FUNCTION_BLOCK TmsEmbarkStation EXTENDS Process IMPLEMENTS ITF_SwitchStation
VAR_INPUT
	StateMachine : IPmlStateMachine;
	TmsSwitch : ITF_TmsSwitch;
END_VAR
VAR_OUTPUT
END_VAR
VAR
	DepartMover : ITmsMover;
	_stationPosition : INT := 1; //1 is low, 2 is high
	State :(
		Init,                                               
		Ready,                                 
        Waiting,
		Processing,
		Register,
		Boarding,
		BoardingComplete,
		Moving); 
	_switchPosition: MC_LREAL;
	demandPosition : SwitchState;
END_VAR

CASE State OF
	Init:
		_Operating := _Clear := _Complete := _Ready := _HasMover := FALSE;
		_Positions[1] := _Positions[2] := _Positions[3] := _Positions[4] := 0;
		NumberOfPositions := 0;
		AssignedPositions := 1;
		StationMovers := 0;
		State := Ready;
	
	Ready:	
		IF StateMachine.GetCurrentState() = E_PMLState.ePMLState_Clearing THEN
			_Operating := _Complete := _HasMover := FALSE;
			_Clear := _Ready := TRUE;
			StationMovers := 0;
			State := Waiting;
		END_IF
	
	Waiting:
		IF _HasMover THEN
			State := Processing;
			_Operating := TRUE;
			_Clear := FALSE;
			_Ready := FALSE;
			_Complete := FALSE;
		END_IF
		
	Processing:
		IF _stationPosition = 1 THEN
			IF TmsSwitch.Switch = SwitchState.Down THEN
				IF DepartMover.ActiveTrack = 16#01010790 THEN
					State := Register;
				ELSE
					DepartMover.ActivateTrack(16#01010790);
					State := Register;
				END_IF
				demandPosition := SwitchState.Middle;
			ELSIF TmsSwitch.Switch = SwitchState.Middle THEN
				IF DepartMover.ActiveTrack = 16#010100E0 THEN
					State := Register;
				ELSE
					DepartMover.ActivateTrack(16#010100E0);
					State := Register;
				END_IF
				demandPosition := SwitchState.Up;
			END_IF
		ELSE
			IF TmsSwitch.Switch = SwitchState.Up THEN
				IF DepartMover.ActiveTrack = 16#010100D0 THEN
					State := Register;
				ELSE
					DepartMover.ActivateTrack(16#010100D0);
					State := Register;
				END_IF
				demandPosition := SwitchState.Middle;
			ELSIF TmsSwitch.Switch = SwitchState.Middle THEN
				IF DepartMover.ActiveTrack = 16#010100F0 THEN
					State := Register;
				ELSE
					DepartMover.ActivateTrack(16#010100F0);
					State := Register;
				END_IF
				demandPosition := SwitchState.Down;
			END_IF
		END_IF
		
	Register:
		TmsSwitch.ExchangeMover(Mover := DepartMover, currentStation := THIS^);
		State := Boarding;
	
	Boarding:
		DepartMover.MoveTo(Position := _switchPosition, Velocity := 100, BackwardMove := FALSE);
		IF DepartMover.isAtPosition(position := _switchPosition) THEN
			State := BoardingComplete;
		END_IF
		
	BoardingComplete:
		IF TmsSwitch.MoveTo(positionState := demandPosition) THEN
			State := Moving;
		END_IF
		
	Moving:
		IF _Complete THEN
			_Operating := FALSE;
			_Clear := TRUE;
			_Ready := TRUE;
			State := Waiting;
		END_IF		
END_CASE

METHOD HasMover : BOOL
VAR_INPUT
	mover : IMover;
END_VAR
VAR
	iTmsMover : ITmsMover;
END_VAR
IF StationMovers <= 2 THEN
	StationMovers := StationMovers + 1;
	IF __QUERYINTERFACE(mover,iTmsMover) THEN
		DepartMover := iTmsMover;
		_HasMover := true;
	END_IF
END_IF
END_METHOD

METHOD PUBLIC MoverAway : BOOL
VAR_INPUT
END_VAR
StationMovers := StationMovers - 1;
DepartMover := 0;
END_METHOD

{warning 'add property implementation'}
PROPERTY StationPosition : INT
GET
StationPosition := _stationPosition;
END_GET
SET
_stationPosition := StationPosition;
END_SET
END_PROPERTY

METHOD PUBLIC SwitchMoveComplete : BOOL
VAR_INPUT
END_VAR
_Complete := SwitchMoveComplete := true;
END_METHOD

{warning 'add property implementation'}
PROPERTY SwitchPosition : mc_lreal
GET
SwitchPosition := _switchPosition;
END_GET
SET
_switchPosition := SwitchPosition;
END_SET
END_PROPERTY

END_FUNCTION_BLOCK

(* stored: Version 1.1.0.1, ProductVersion 3.1.4024.11
   POU TmsEmbarkStation: Id {044d9b9f-48a1-452d-b127-28199a3c04bb}, SpecialFunc None
   Method HasMover: Id {6096dfca-b0c2-4998-b7bb-2c09860d3176}
   Method MoverAway: Id {5d30fab5-165d-4159-bdc5-36df29db049b}
   Property StationPosition: Id {04b01043-8abc-480b-b7a1-3b47b2f6b3d3}
   Get Get: Id {63f29fcb-9246-41b7-8237-0e14a4d877b8}
   Set Set: Id {8dad77b7-b3d3-4e11-af0a-1ace0eb16549}
   Method SwitchMoveComplete: Id {b6e4018d-1b11-4436-abf3-c2d1900106a2}
   Property SwitchPosition: Id {77eb7d82-50db-4968-86fb-d2f009644fbf}
   Get Get: Id {5e9136b4-3bc6-41b5-a233-22f210e01c6b}
   Set Set: Id {58d1b30d-be8b-4b08-b209-84e887ca28ad} *)
